TYPE ST_TUR_6_0 :
(**************************************************************************************
 * 	Application		:	BoxControl Framework
 *	Revision		:	$Revision: 404529 $
 *	Revision date	:	$Date: 2018-04-23 08:21:38 +0200 (Mo., 23 Apr 2018) $
 *	Last changed by	:	$Author: b7bolm $
 *	URL				:	$URL: http://almscdc.swisslog.com/repo/SWPD/Development/BoxControlFramework/20_Release/trunk/01_Software/BCF/BCF/JumpStart/20_Product/10_App/11_Com/10_Lib/10_Conv/12_MFCS/11_SIS/01_DUTs/10_SIS_6_0/ST_TUR_6_0.TcDUT $
 *
 *	Purpose			:	TTQ Structure
 *
 * ------------------------------------------------------------------------------------
 *	Copyright Swisslog [IP AG], Switzerland. All rights reserved.
 * 
 * ------------------------------------------------------------------------------------
 *	
 * 	Revision History: 
 *
 * 	VERSION			DATE			INITIALS			DESCRIPTION
 *	0.1				01.01.2001		swl					Example
 *
 **************************************************************************************)
STRUCT
	Position				: STRING(SIS_6_0.POSITION_STRINGLENGTH); // 12 Digit SIS Location MM-GGG-EEEE-FF-Z 
	TU_DataIndex			: STRING(SIS_6_0.TU_DATAINDEX_STRINGLENGTH); // 6 Digit Tu Index
	TU_ID					: STRING(SIS_6_0.TU_ID_STRINGLENGTH); // 18 Digit SSID 
	TU_Type					: STRING(SIS_6_0.TU_TYPE_STRINGLENGTH); // 2 Digit of type
	AssignmentID			: STRING(SIS_6_0.ASSIGNMENT_ID_STRINGLENGTH); // 8 Assignment
	Length					: STRING(SIS_6_0.DIMENSIONS); // 4 Digit dimension
	Width					: STRING(SIS_6_0.DIMENSIONS); // 4 Digit dimension
	Height					: STRING(SIS_6_0.DIMENSIONS); // 4 Digit dimension
	Weight					: STRING(SIS_6_0.TTA_WEIGHT); // 8 Digit weight
	Orientation				: STRING(SIS_6_0.TTA_ORIENTATION);
	TU_Parameter 			: STRING(SIS_6_0.TTA_TU_PARAMETER); // 4 Digit parameter
	IO_Data					: STRING(SIS_6_0.TUR_IO_DATA_STRINGLENGTH); (* 3 Digit IO Data *)
	LowerLimit				: STRING(SIS_6_0.TUR_LOWERLIMIT_STRINGLENGTH); (* 7 Digit Lower Limit *)
	UpperLimit				: STRING(SIS_6_0.TUR_UPPERLIMIT_STRINGLENGTH); (* 7 Digit Upper Limit *)
	GroupInfo				: STRING(SIS_6_0.TUR_GROUPINFO_STRINGLENGTH); (* 4 Digit Group Information *)
	Sequence				: STRING(SIS_6_0.TUR_SEQUENCE_STRINGLENGTH); (* 4 Digit Sequence Number *)
	NumberInSequence		: STRING(SIS_6_0.TUR_NUMBER_IN_SEQUENCE_STRINGLENGTH); (* 4 Digit Number in Sequence *)
	ReturnCode				: STRING(SIS_6_0.ERRORCODE_STRINGLENGTH); // 4 Digit return code
	NumberOfDestinations	: STRING(SIS_6_0.TUR_NUMBER_OF_DESTINATIONS_STRINGLENGTH); (* 2 Digit Number of Destinations *)
	Destination				: ARRAY [1..99] OF STRING(SIS_6_0.POSITION_STRINGLENGTH); (* Array of 12 Digit SIS Destinations *)
END_STRUCT
END_TYPE

(* stored: Version 1.1.0.1, ProductVersion 3.1.4022.12
   DUT ST_TUR_6_0: Id {ce02f79e-6478-4c5a-905b-038ad0aaf8c5} *)
